Staubli VAL3: runLow.pgx

public program runLow()
begin
  if data:setDryRun==true
    if SYS:diMachineInAuto[moduleIndex]==true
      data:setDryRun=false
      call scr:popUp("Dry run mode automatically deactivated because IMM is in 'Automatic' mode!",data:nMsgTimeOut,false)
    endIf
    if bRobotOff==true
      data:setDryRun=false
      call scr:popUp("Dry run mode automatically deactivated because robot is disabled!",data:nMsgTimeOut,false)
    endIf
  endIf
end
